// TIA Portal V15.1 export
// export: Created 2024-05-17T05:38:54.7838855Z, ExportSetting WithDefaults, DisplayName Totally Integrated Automation Portal, DisplayVersion V15.1 Update 5, DisplayName TIA Portal Openness, DisplayVersion V15.1 Update 5, DisplayName SINAMICS Startdrive Advanced, DisplayVersion V15.1, DisplayName G130, G150, S120, S150, SINAMICS MV, S210, DisplayVersion V15.1, DisplayName G110M, G120, G120C, G120D, G120P, DisplayVersion V15.1, DisplayName STEP 7 Professional, DisplayVersion V15.1 Update 5, DisplayName STEP 7 Safety, DisplayVersion V15.1, DisplayName WinCC Professional, DisplayVersion V15.1 Update 5, DisplayName SIMATIC Visualization Architect, DisplayVersion V15.1
FUNCTION "209220ZS01Safety" : Void   // FC375, FBD
TITLE = 209220ZS01 Safety
{ S7_Optimized_Access := 'FALSE' }
AUTHOR : VCG
FAMILY : Local
NAME : 610
VERSION : 0.1
// stored: AutoNumber false, IsIECCheckEnabled false, SetENOAutomatically False, UDAEnableTagReadback false
   VAR_OUTPUT
      O_AlarmA : Bool;   // Alarm A
      O_AlarmB : Bool;   // Alarm B
      O_AlarmC : Bool;   // Alarm C
      O_AlarmD : Bool;   // Alarm D
      O_AlarmABCondition : Bool;   // Alarms resetable
      H_IAnim : Word;   // Icon Animation
   END_VAR
BEGIN

REGION Network 1: **** 2.1 - Enable Alarms **** 220CS22M4SG10F & SG11F Check if both safety sensors are activated
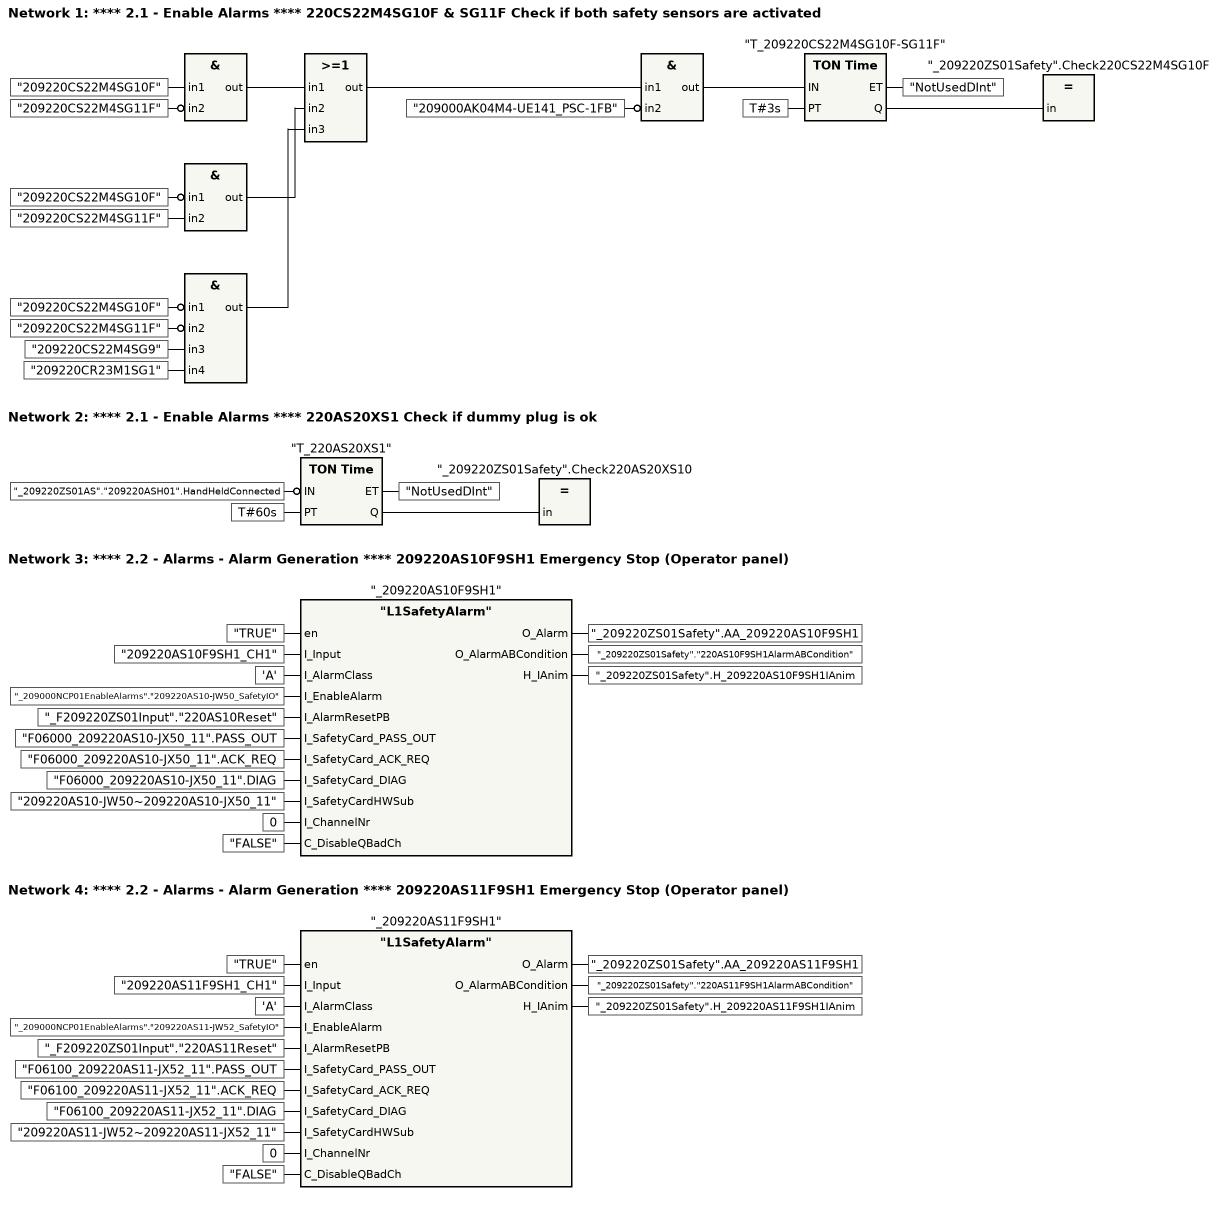
   "T_209220CS22M4SG10F-SG11F".TON(IN := (("209220CS22M4SG10F" AND NOT "209220CS22M4SG11F") OR (NOT "209220CS22M4SG10F" AND "209220CS22M4SG11F") OR (NOT "209220CS22M4SG10F" AND NOT "209220CS22M4SG11F" AND "209220CS22M4SG9" AND "209220CR23M1SG1")) AND NOT "209000AK04M4-UE141_PSC-1FB",
                           PT := T#3s,
                           ET => "NotUsedDInt");
   "_209220ZS01Safety".Check220CS22M4SG10F := "T_209220CS22M4SG10F-SG11F".Q;
END_REGION

REGION Network 2: **** 2.1 - Enable Alarms **** 220AS20XS1 Check if dummy plug is ok
   "T_220AS20XS1".TON(IN := NOT "_209220ZS01AS"."209220ASH01".HandHeldConnected,
                      PT := T#60s,
                      ET => "NotUsedDInt");
   "_209220ZS01Safety".Check220AS20XS10 := "T_220AS20XS1".Q;
END_REGION

REGION Network 3: **** 2.2 - Alarms - Alarm Generation **** 209220AS10F9SH1 Emergency Stop (Operator panel)
   // Emergency Stop
   IF "TRUE" THEN
       "_209220AS10F9SH1"(I_Input := "209220AS10F9SH1_CH1",   // "L1SafetyAlarm"
                          I_AlarmClass := 'A',
                          I_EnableAlarm := "_209000NCP01EnableAlarms"."209220AS10-JW50_SafetyIO",
                          I_AlarmResetPB := "_F209220ZS01Input"."220AS10Reset",
                          I_SafetyCard_PASS_OUT := "F06000_209220AS10-JX50_11".PASS_OUT,
                          I_SafetyCard_ACK_REQ := "F06000_209220AS10-JX50_11".ACK_REQ,
                          I_SafetyCard_DIAG := "F06000_209220AS10-JX50_11".DIAG,
                          I_SafetyCardHWSub := "209220AS10-JW50~209220AS10-JX50_11",
                          I_ChannelNr := 0,
                          C_DisableQBadCh := "FALSE",
                          O_Alarm => "_209220ZS01Safety".AA_209220AS10F9SH1,
                          O_AlarmABCondition => "_209220ZS01Safety"."220AS10F9SH1AlarmABCondition",
                          H_IAnim => "_209220ZS01Safety".H_209220AS10F9SH1IAnim);
   END_IF;
END_REGION

REGION Network 4: **** 2.2 - Alarms - Alarm Generation **** 209220AS11F9SH1 Emergency Stop (Operator panel)
   // Emergency Stop
   IF "TRUE" THEN
       "_209220AS11F9SH1"(I_Input := "209220AS11F9SH1_CH1",   // "L1SafetyAlarm"
                          I_AlarmClass := 'A',
                          I_EnableAlarm := "_209000NCP01EnableAlarms"."209220AS11-JW52_SafetyIO",
                          I_AlarmResetPB := "_F209220ZS01Input"."220AS11Reset",
                          I_SafetyCard_PASS_OUT := "F06100_209220AS11-JX52_11".PASS_OUT,
                          I_SafetyCard_ACK_REQ := "F06100_209220AS11-JX52_11".ACK_REQ,
                          I_SafetyCard_DIAG := "F06100_209220AS11-JX52_11".DIAG,
                          I_SafetyCardHWSub := "209220AS11-JW52~209220AS11-JX52_11",
                          I_ChannelNr := 0,
                          C_DisableQBadCh := "FALSE",
                          O_Alarm => "_209220ZS01Safety".AA_209220AS11F9SH1,
                          O_AlarmABCondition => "_209220ZS01Safety"."220AS11F9SH1AlarmABCondition",
                          H_IAnim => "_209220ZS01Safety".H_209220AS11F9SH1IAnim);
   END_IF;
END_REGION

REGION Network 5: **** 2.2 - Alarms - Alarm Generation **** 209220AS20F9SH1 Emergency Stop (Start/Stop panel)
   // Emergency Stop
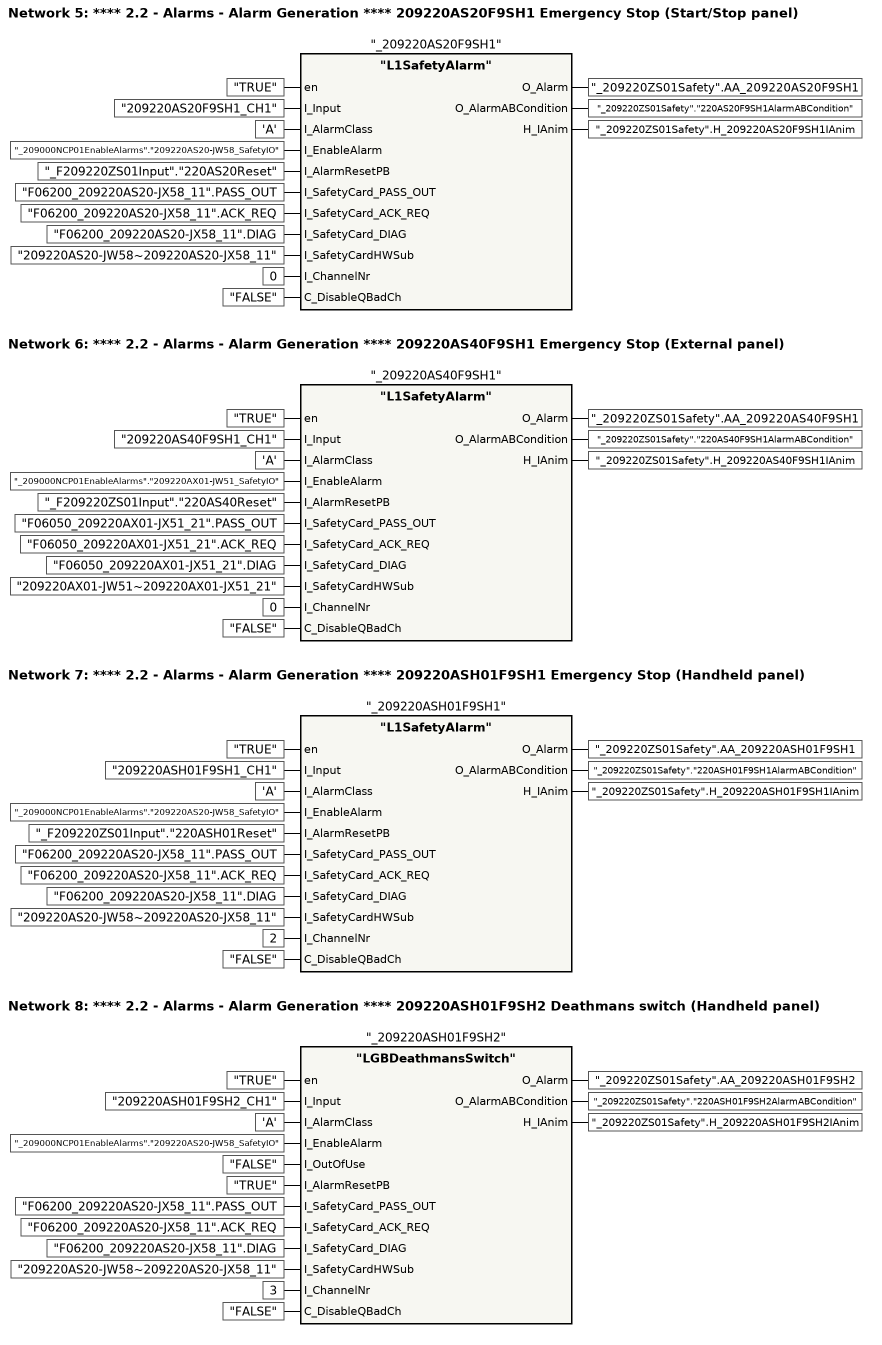
   IF "TRUE" THEN
       "_209220AS20F9SH1"(I_Input := "209220AS20F9SH1_CH1",   // "L1SafetyAlarm"
                          I_AlarmClass := 'A',
                          I_EnableAlarm := "_209000NCP01EnableAlarms"."209220AS20-JW58_SafetyIO",
                          I_AlarmResetPB := "_F209220ZS01Input"."220AS20Reset",
                          I_SafetyCard_PASS_OUT := "F06200_209220AS20-JX58_11".PASS_OUT,
                          I_SafetyCard_ACK_REQ := "F06200_209220AS20-JX58_11".ACK_REQ,
                          I_SafetyCard_DIAG := "F06200_209220AS20-JX58_11".DIAG,
                          I_SafetyCardHWSub := "209220AS20-JW58~209220AS20-JX58_11",
                          I_ChannelNr := 0,
                          C_DisableQBadCh := "FALSE",
                          O_Alarm => "_209220ZS01Safety".AA_209220AS20F9SH1,
                          O_AlarmABCondition => "_209220ZS01Safety"."220AS20F9SH1AlarmABCondition",
                          H_IAnim => "_209220ZS01Safety".H_209220AS20F9SH1IAnim);
   END_IF;
END_REGION

REGION Network 6: **** 2.2 - Alarms - Alarm Generation **** 209220AS40F9SH1 Emergency Stop (External panel)
   // Emergency Stop
   IF "TRUE" THEN
       "_209220AS40F9SH1"(I_Input := "209220AS40F9SH1_CH1",   // "L1SafetyAlarm"
                          I_AlarmClass := 'A',
                          I_EnableAlarm := "_209000NCP01EnableAlarms"."209220AX01-JW51_SafetyIO",
                          I_AlarmResetPB := "_F209220ZS01Input"."220AS40Reset",
                          I_SafetyCard_PASS_OUT := "F06050_209220AX01-JX51_21".PASS_OUT,
                          I_SafetyCard_ACK_REQ := "F06050_209220AX01-JX51_21".ACK_REQ,
                          I_SafetyCard_DIAG := "F06050_209220AX01-JX51_21".DIAG,
                          I_SafetyCardHWSub := "209220AX01-JW51~209220AX01-JX51_21",
                          I_ChannelNr := 0,
                          C_DisableQBadCh := "FALSE",
                          O_Alarm => "_209220ZS01Safety".AA_209220AS40F9SH1,
                          O_AlarmABCondition => "_209220ZS01Safety"."220AS40F9SH1AlarmABCondition",
                          H_IAnim => "_209220ZS01Safety".H_209220AS40F9SH1IAnim);
   END_IF;
END_REGION

REGION Network 7: **** 2.2 - Alarms - Alarm Generation **** 209220ASH01F9SH1 Emergency Stop (Handheld panel)
   // Emergency Stop
   IF "TRUE" THEN
       "_209220ASH01F9SH1"(I_Input := "209220ASH01F9SH1_CH1",   // "L1SafetyAlarm"
                           I_AlarmClass := 'A',
                           I_EnableAlarm := "_209000NCP01EnableAlarms"."209220AS20-JW58_SafetyIO",
                           I_AlarmResetPB := "_F209220ZS01Input"."220ASH01Reset",
                           I_SafetyCard_PASS_OUT := "F06200_209220AS20-JX58_11".PASS_OUT,
                           I_SafetyCard_ACK_REQ := "F06200_209220AS20-JX58_11".ACK_REQ,
                           I_SafetyCard_DIAG := "F06200_209220AS20-JX58_11".DIAG,
                           I_SafetyCardHWSub := "209220AS20-JW58~209220AS20-JX58_11",
                           I_ChannelNr := 2,
                           C_DisableQBadCh := "FALSE",
                           O_Alarm => "_209220ZS01Safety".AA_209220ASH01F9SH1,
                           O_AlarmABCondition => "_209220ZS01Safety"."220ASH01F9SH1AlarmABCondition",
                           H_IAnim => "_209220ZS01Safety".H_209220ASH01F9SH1IAnim);
   END_IF;
END_REGION

REGION Network 8: **** 2.2 - Alarms - Alarm Generation **** 209220ASH01F9SH2 Deathmans switch (Handheld panel)
   // Deathmans switch
   IF "TRUE" THEN
       "_209220ASH01F9SH2"(I_Input := "209220ASH01F9SH2_CH1",   // "LGBDeathmansSwitch"
                           I_AlarmClass := 'A',
                           I_EnableAlarm := "_209000NCP01EnableAlarms"."209220AS20-JW58_SafetyIO",
                           I_OutOfUse := "FALSE",
                           I_AlarmResetPB := "TRUE",
                           I_SafetyCard_PASS_OUT := "F06200_209220AS20-JX58_11".PASS_OUT,
                           I_SafetyCard_ACK_REQ := "F06200_209220AS20-JX58_11".ACK_REQ,
                           I_SafetyCard_DIAG := "F06200_209220AS20-JX58_11".DIAG,
                           I_SafetyCardHWSub := "209220AS20-JW58~209220AS20-JX58_11",
                           I_ChannelNr := 3,
                           C_DisableQBadCh := "FALSE",
                           O_Alarm => "_209220ZS01Safety".AA_209220ASH01F9SH2,
                           O_AlarmABCondition => "_209220ZS01Safety"."220ASH01F9SH2AlarmABCondition",
                           H_IAnim => "_209220ZS01Safety".H_209220ASH01F9SH2IAnim);
   END_IF;
END_REGION

REGION Network 9: **** 2.2 - Alarms - Alarm Generation **** 020R02F9SH / **** 2.2 - Alarms - Alarm Generation **** 209000AK04F9QC1FB Feedback Alarm
   // E-Stop Push Button / Feedback Alarm
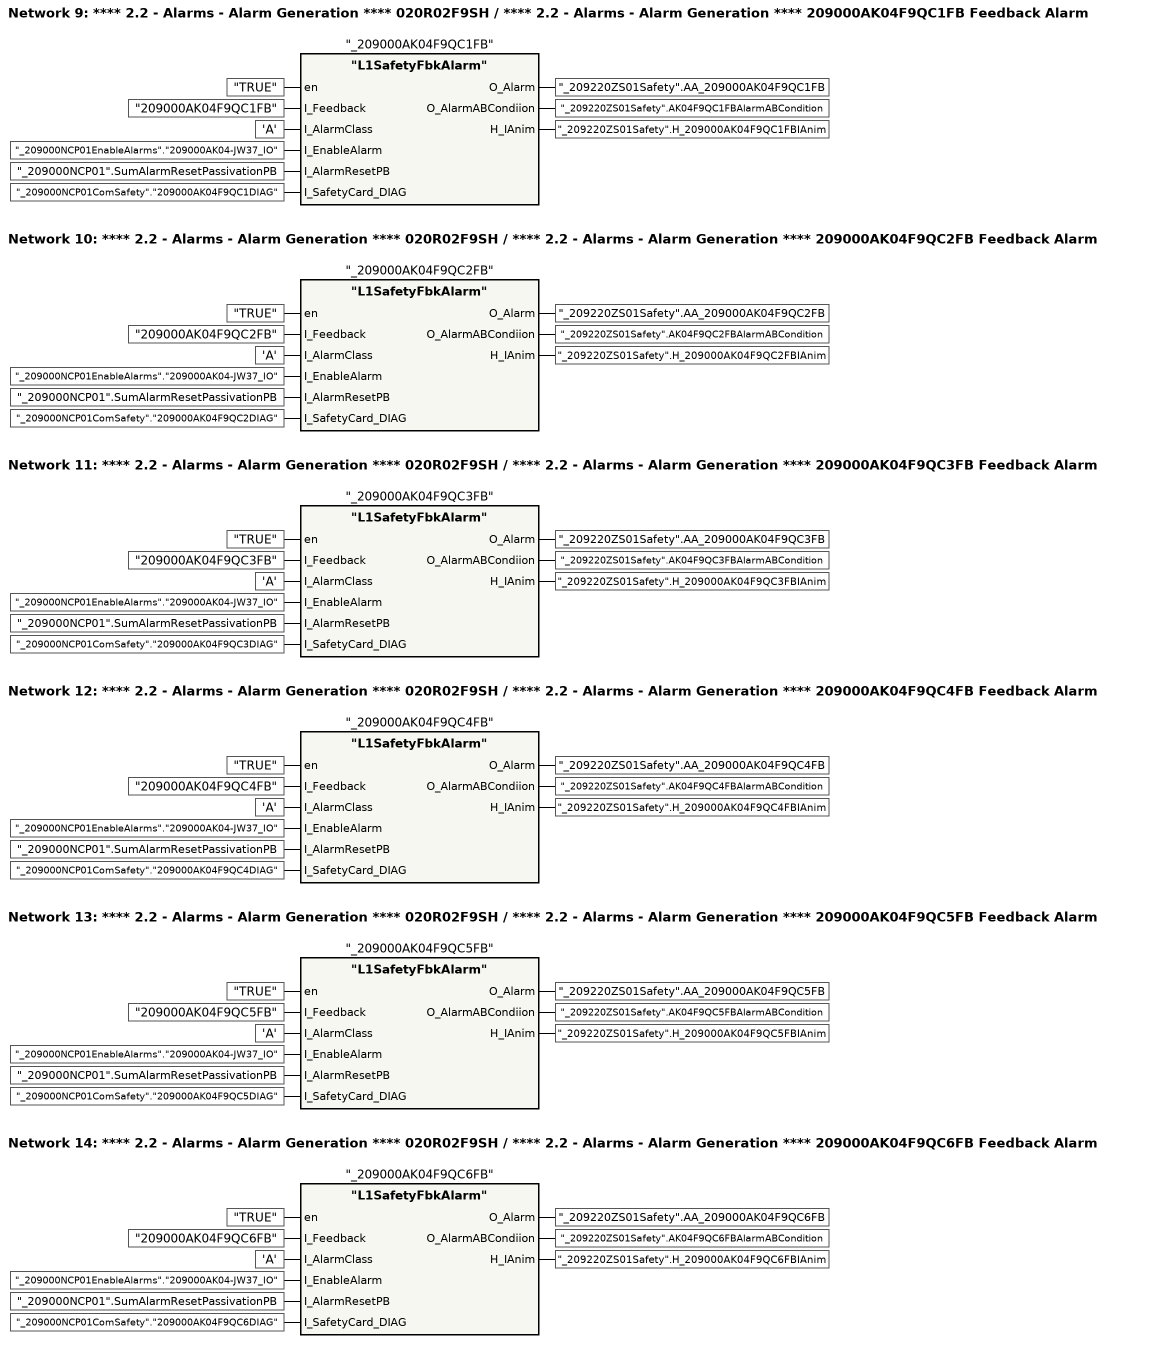
   IF "TRUE" THEN
       "_209000AK04F9QC1FB"(I_Feedback := "209000AK04F9QC1FB",   // "L1SafetyFbkAlarm"
                            I_AlarmClass := 'A',
                            I_EnableAlarm := "_209000NCP01EnableAlarms"."209000AK04-JW37_IO",
                            I_AlarmResetPB := "_209000NCP01".SumAlarmResetPassivationPB,
                            I_SafetyCard_DIAG := "_209000NCP01ComSafety"."209000AK04F9QC1DIAG",
                            O_Alarm => "_209220ZS01Safety".AA_209000AK04F9QC1FB,
                            O_AlarmABCondiion => "_209220ZS01Safety".AK04F9QC1FBAlarmABCondition,
                            H_IAnim => "_209220ZS01Safety".H_209000AK04F9QC1FBIAnim);
   END_IF;
END_REGION

REGION Network 10: **** 2.2 - Alarms - Alarm Generation **** 020R02F9SH / **** 2.2 - Alarms - Alarm Generation **** 209000AK04F9QC2FB Feedback Alarm
   // E-Stop Push Button / Feedback Alarm
   IF "TRUE" THEN
       "_209000AK04F9QC2FB"(I_Feedback := "209000AK04F9QC2FB",   // "L1SafetyFbkAlarm"
                            I_AlarmClass := 'A',
                            I_EnableAlarm := "_209000NCP01EnableAlarms"."209000AK04-JW37_IO",
                            I_AlarmResetPB := "_209000NCP01".SumAlarmResetPassivationPB,
                            I_SafetyCard_DIAG := "_209000NCP01ComSafety"."209000AK04F9QC2DIAG",
                            O_Alarm => "_209220ZS01Safety".AA_209000AK04F9QC2FB,
                            O_AlarmABCondiion => "_209220ZS01Safety".AK04F9QC2FBAlarmABCondition,
                            H_IAnim => "_209220ZS01Safety".H_209000AK04F9QC2FBIAnim);
   END_IF;
END_REGION

REGION Network 11: **** 2.2 - Alarms - Alarm Generation **** 020R02F9SH / **** 2.2 - Alarms - Alarm Generation **** 209000AK04F9QC3FB Feedback Alarm
   // E-Stop Push Button / Feedback Alarm
   IF "TRUE" THEN
       "_209000AK04F9QC3FB"(I_Feedback := "209000AK04F9QC3FB",   // "L1SafetyFbkAlarm"
                            I_AlarmClass := 'A',
                            I_EnableAlarm := "_209000NCP01EnableAlarms"."209000AK04-JW37_IO",
                            I_AlarmResetPB := "_209000NCP01".SumAlarmResetPassivationPB,
                            I_SafetyCard_DIAG := "_209000NCP01ComSafety"."209000AK04F9QC3DIAG",
                            O_Alarm => "_209220ZS01Safety".AA_209000AK04F9QC3FB,
                            O_AlarmABCondiion => "_209220ZS01Safety".AK04F9QC3FBAlarmABCondition,
                            H_IAnim => "_209220ZS01Safety".H_209000AK04F9QC3FBIAnim);
   END_IF;
END_REGION

REGION Network 12: **** 2.2 - Alarms - Alarm Generation **** 020R02F9SH / **** 2.2 - Alarms - Alarm Generation **** 209000AK04F9QC4FB Feedback Alarm
   // E-Stop Push Button / Feedback Alarm
   IF "TRUE" THEN
       "_209000AK04F9QC4FB"(I_Feedback := "209000AK04F9QC4FB",   // "L1SafetyFbkAlarm"
                            I_AlarmClass := 'A',
                            I_EnableAlarm := "_209000NCP01EnableAlarms"."209000AK04-JW37_IO",
                            I_AlarmResetPB := "_209000NCP01".SumAlarmResetPassivationPB,
                            I_SafetyCard_DIAG := "_209000NCP01ComSafety"."209000AK04F9QC4DIAG",
                            O_Alarm => "_209220ZS01Safety".AA_209000AK04F9QC4FB,
                            O_AlarmABCondiion => "_209220ZS01Safety".AK04F9QC4FBAlarmABCondition,
                            H_IAnim => "_209220ZS01Safety".H_209000AK04F9QC4FBIAnim);
   END_IF;
END_REGION

REGION Network 13: **** 2.2 - Alarms - Alarm Generation **** 020R02F9SH / **** 2.2 - Alarms - Alarm Generation **** 209000AK04F9QC5FB Feedback Alarm
   // E-Stop Push Button / Feedback Alarm
   IF "TRUE" THEN
       "_209000AK04F9QC5FB"(I_Feedback := "209000AK04F9QC5FB",   // "L1SafetyFbkAlarm"
                            I_AlarmClass := 'A',
                            I_EnableAlarm := "_209000NCP01EnableAlarms"."209000AK04-JW37_IO",
                            I_AlarmResetPB := "_209000NCP01".SumAlarmResetPassivationPB,
                            I_SafetyCard_DIAG := "_209000NCP01ComSafety"."209000AK04F9QC5DIAG",
                            O_Alarm => "_209220ZS01Safety".AA_209000AK04F9QC5FB,
                            O_AlarmABCondiion => "_209220ZS01Safety".AK04F9QC5FBAlarmABCondition,
                            H_IAnim => "_209220ZS01Safety".H_209000AK04F9QC5FBIAnim);
   END_IF;
END_REGION

REGION Network 14: **** 2.2 - Alarms - Alarm Generation **** 020R02F9SH / **** 2.2 - Alarms - Alarm Generation **** 209000AK04F9QC6FB Feedback Alarm
   // E-Stop Push Button / Feedback Alarm
   IF "TRUE" THEN
       "_209000AK04F9QC6FB"(I_Feedback := "209000AK04F9QC6FB",   // "L1SafetyFbkAlarm"
                            I_AlarmClass := 'A',
                            I_EnableAlarm := "_209000NCP01EnableAlarms"."209000AK04-JW37_IO",
                            I_AlarmResetPB := "_209000NCP01".SumAlarmResetPassivationPB,
                            I_SafetyCard_DIAG := "_209000NCP01ComSafety"."209000AK04F9QC6DIAG",
                            O_Alarm => "_209220ZS01Safety".AA_209000AK04F9QC6FB,
                            O_AlarmABCondiion => "_209220ZS01Safety".AK04F9QC6FBAlarmABCondition,
                            H_IAnim => "_209220ZS01Safety".H_209000AK04F9QC6FBIAnim);
   END_IF;
END_REGION

REGION Network 15: **** 2.2 - Alarms - Alarm Generation **** 209220CHB21M14SG1F Safety sensor
   // Safety sensor
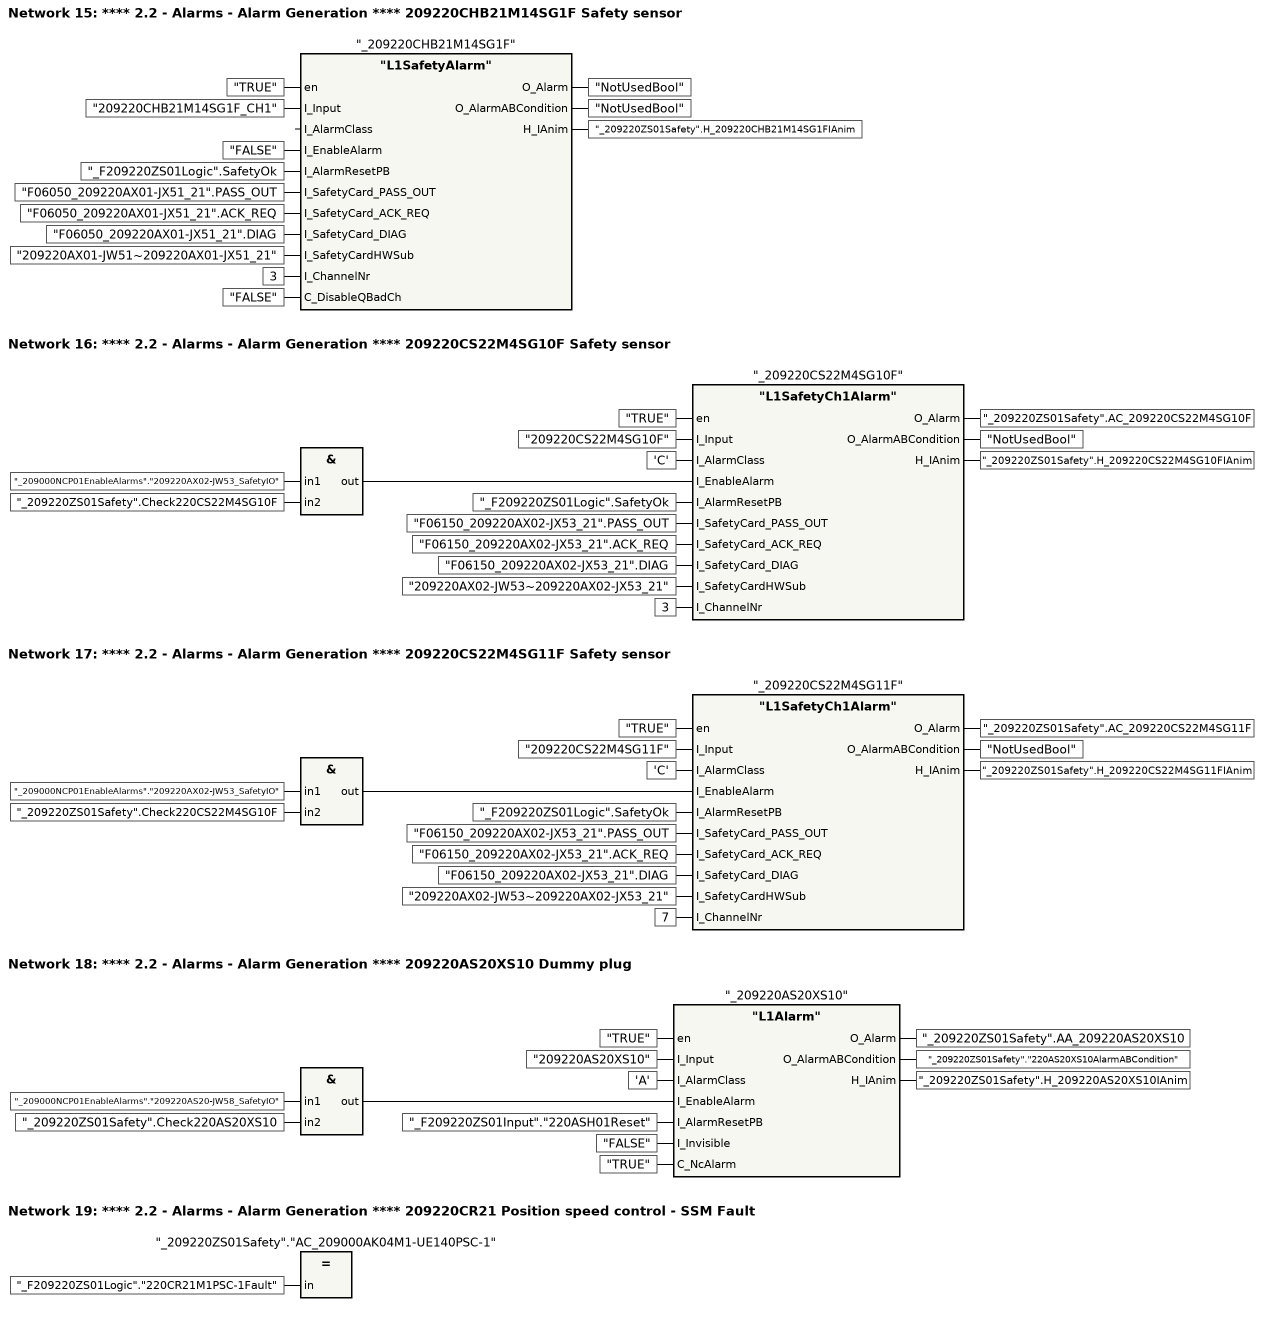
   IF "TRUE" THEN
       "_209220CHB21M14SG1F"(I_Input := "209220CHB21M14SG1F_CH1",   // "L1SafetyAlarm"
                             I_EnableAlarm := "FALSE",
                             I_AlarmResetPB := "_F209220ZS01Logic".SafetyOk,
                             I_SafetyCard_PASS_OUT := "F06050_209220AX01-JX51_21".PASS_OUT,
                             I_SafetyCard_ACK_REQ := "F06050_209220AX01-JX51_21".ACK_REQ,
                             I_SafetyCard_DIAG := "F06050_209220AX01-JX51_21".DIAG,
                             I_SafetyCardHWSub := "209220AX01-JW51~209220AX01-JX51_21",
                             I_ChannelNr := 3,
                             C_DisableQBadCh := "FALSE",
                             O_Alarm => "NotUsedBool",
                             O_AlarmABCondition => "NotUsedBool",
                             H_IAnim => "_209220ZS01Safety".H_209220CHB21M14SG1FIAnim);
   END_IF;
END_REGION

REGION Network 16: **** 2.2 - Alarms - Alarm Generation **** 209220CS22M4SG10F Safety sensor
   // Safety sensor
   IF "TRUE" THEN
       "_209220CS22M4SG10F"(I_Input := "209220CS22M4SG10F",   // "L1SafetyCh1Alarm"
                            I_AlarmClass := 'C',
                            I_EnableAlarm := "_209000NCP01EnableAlarms"."209220AX02-JW53_SafetyIO" AND "_209220ZS01Safety".Check220CS22M4SG10F,
                            I_AlarmResetPB := "_F209220ZS01Logic".SafetyOk,
                            I_SafetyCard_PASS_OUT := "F06150_209220AX02-JX53_21".PASS_OUT,
                            I_SafetyCard_ACK_REQ := "F06150_209220AX02-JX53_21".ACK_REQ,
                            I_SafetyCard_DIAG := "F06150_209220AX02-JX53_21".DIAG,
                            I_SafetyCardHWSub := "209220AX02-JW53~209220AX02-JX53_21",
                            I_ChannelNr := 3,
                            O_Alarm => "_209220ZS01Safety".AC_209220CS22M4SG10F,
                            O_AlarmABCondition => "NotUsedBool",
                            H_IAnim => "_209220ZS01Safety".H_209220CS22M4SG10FIAnim);
   END_IF;
END_REGION

REGION Network 17: **** 2.2 - Alarms - Alarm Generation **** 209220CS22M4SG11F Safety sensor
   // Safety sensor
   IF "TRUE" THEN
       "_209220CS22M4SG11F"(I_Input := "209220CS22M4SG11F",   // "L1SafetyCh1Alarm"
                            I_AlarmClass := 'C',
                            I_EnableAlarm := "_209000NCP01EnableAlarms"."209220AX02-JW53_SafetyIO" AND "_209220ZS01Safety".Check220CS22M4SG10F,
                            I_AlarmResetPB := "_F209220ZS01Logic".SafetyOk,
                            I_SafetyCard_PASS_OUT := "F06150_209220AX02-JX53_21".PASS_OUT,
                            I_SafetyCard_ACK_REQ := "F06150_209220AX02-JX53_21".ACK_REQ,
                            I_SafetyCard_DIAG := "F06150_209220AX02-JX53_21".DIAG,
                            I_SafetyCardHWSub := "209220AX02-JW53~209220AX02-JX53_21",
                            I_ChannelNr := 7,
                            O_Alarm => "_209220ZS01Safety".AC_209220CS22M4SG11F,
                            O_AlarmABCondition => "NotUsedBool",
                            H_IAnim => "_209220ZS01Safety".H_209220CS22M4SG11FIAnim);
   END_IF;
END_REGION

REGION Network 18: **** 2.2 - Alarms - Alarm Generation **** 209220AS20XS10 Dummy plug
   IF "TRUE" THEN
       "_209220AS20XS10"(I_Input := "209220AS20XS10",   // "L1Alarm"
                         I_AlarmClass := 'A',
                         I_EnableAlarm := "_209000NCP01EnableAlarms"."209220AS20-JW58_SafetyIO" AND "_209220ZS01Safety".Check220AS20XS10,
                         I_AlarmResetPB := "_F209220ZS01Input"."220ASH01Reset",
                         I_Invisible := "FALSE",
                         C_NcAlarm := "TRUE",
                         O_Alarm => "_209220ZS01Safety".AA_209220AS20XS10,
                         O_AlarmABCondition => "_209220ZS01Safety"."220AS20XS10AlarmABCondition",
                         H_IAnim => "_209220ZS01Safety".H_209220AS20XS10IAnim);
   END_IF;
END_REGION

REGION Network 19: **** 2.2 - Alarms - Alarm Generation **** 209220CR21 Position speed control - SSM Fault
   // SEW Safety Function
   "_209220ZS01Safety"."AC_209000AK04M1-UE140PSC-1" := "_F209220ZS01Logic"."220CR21M1PSC-1Fault";
END_REGION

REGION Network 20: **** 2.2 - Alarms - Alarm Generation **** 209220CS22 Position speed control - SSM Fault
   // SEW Safety Function
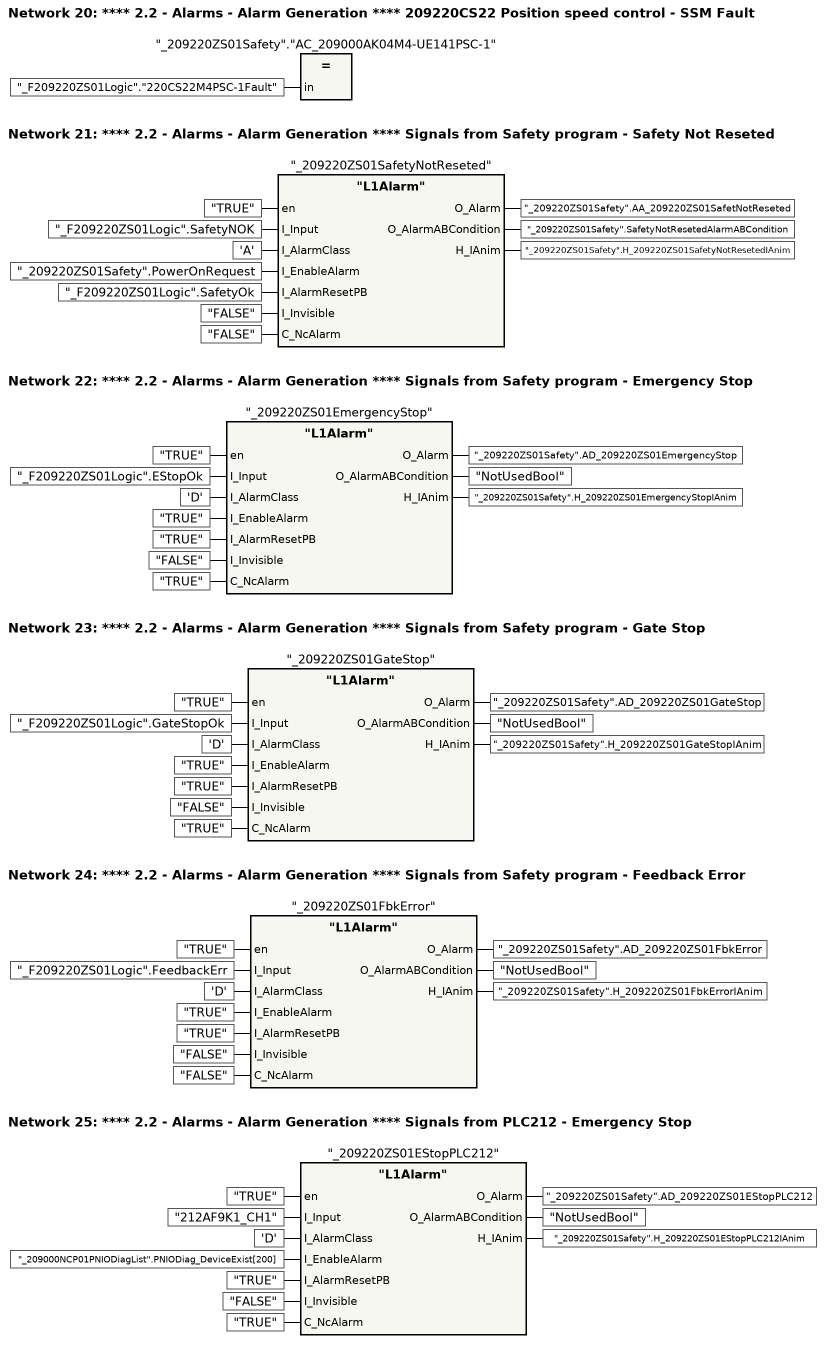
   "_209220ZS01Safety"."AC_209000AK04M4-UE141PSC-1" := "_F209220ZS01Logic"."220CS22M4PSC-1Fault";
END_REGION

REGION Network 21: **** 2.2 - Alarms - Alarm Generation **** Signals from Safety program - Safety Not Reseted
   // Safety Has Not Been Reseted
   IF "TRUE" THEN
       "_209220ZS01SafetyNotReseted"(I_Input := "_F209220ZS01Logic".SafetyNOK,   // "L1Alarm"
                               I_AlarmClass := 'A',
                               I_EnableAlarm := "_209220ZS01Safety".PowerOnRequest,
                               I_AlarmResetPB := "_F209220ZS01Logic".SafetyOk,
                               I_Invisible := "FALSE",
                               C_NcAlarm := "FALSE",
                               O_Alarm => "_209220ZS01Safety".AA_209220ZS01SafetNotReseted,
                               O_AlarmABCondition => "_209220ZS01Safety".SafetyNotResetedAlarmABCondition,
                               H_IAnim => "_209220ZS01Safety".H_209220ZS01SafetyNotResetedIAnim);
   END_IF;
END_REGION

REGION Network 22: **** 2.2 - Alarms - Alarm Generation **** Signals from Safety program - Emergency Stop
   // Emergency Stop
   IF "TRUE" THEN
       "_209220ZS01EmergencyStop"(I_Input := "_F209220ZS01Logic".EStopOk,   // "L1Alarm"
                               I_AlarmClass := 'D',
                               I_EnableAlarm := "TRUE",
                               I_AlarmResetPB := "TRUE",
                               I_Invisible := "FALSE",
                               C_NcAlarm := "TRUE",
                               O_Alarm => "_209220ZS01Safety".AD_209220ZS01EmergencyStop,
                               O_AlarmABCondition => "NotUsedBool",
                               H_IAnim => "_209220ZS01Safety".H_209220ZS01EmergencyStopIAnim);
   END_IF;
END_REGION

REGION Network 23: **** 2.2 - Alarms - Alarm Generation **** Signals from Safety program - Gate Stop
   // Gate Stop
   IF "TRUE" THEN
       "_209220ZS01GateStop"(I_Input := "_F209220ZS01Logic".GateStopOk,   // "L1Alarm"
                             I_AlarmClass := 'D',
                             I_EnableAlarm := "TRUE",
                             I_AlarmResetPB := "TRUE",
                             I_Invisible := "FALSE",
                             C_NcAlarm := "TRUE",
                             O_Alarm => "_209220ZS01Safety".AD_209220ZS01GateStop,
                             O_AlarmABCondition => "NotUsedBool",
                             H_IAnim => "_209220ZS01Safety".H_209220ZS01GateStopIAnim);
   END_IF;
END_REGION

REGION Network 24: **** 2.2 - Alarms - Alarm Generation **** Signals from Safety program - Feedback Error
   // Feedback Error
   IF "TRUE" THEN
       "_209220ZS01FbkError"(I_Input := "_F209220ZS01Logic".FeedbackErr,   // "L1Alarm"
                             I_AlarmClass := 'D',
                             I_EnableAlarm := "TRUE",
                             I_AlarmResetPB := "TRUE",
                             I_Invisible := "FALSE",
                             C_NcAlarm := "FALSE",
                             O_Alarm => "_209220ZS01Safety".AD_209220ZS01FbkError,
                             O_AlarmABCondition => "NotUsedBool",
                             H_IAnim => "_209220ZS01Safety".H_209220ZS01FbkErrorIAnim);
   END_IF;
END_REGION

REGION Network 25: **** 2.2 - Alarms - Alarm Generation **** Signals from PLC212 - Emergency Stop
   IF "TRUE" THEN
       "_209220ZS01EStopPLC212"(I_Input := "212AF9K1_CH1",   // "L1Alarm"
                               I_AlarmClass := 'D',
                               I_EnableAlarm := "_209000NCP01PNIODiagList".PNIODiag_DeviceExist[200],
                               I_AlarmResetPB := "TRUE",
                               I_Invisible := "FALSE",
                               C_NcAlarm := "TRUE",
                               O_Alarm => "_209220ZS01Safety".AD_209220ZS01EStopPLC212,
                               O_AlarmABCondition => "NotUsedBool",
                               H_IAnim => "_209220ZS01Safety".H_209220ZS01EStopPLC212IAnim);
   END_IF;
END_REGION

REGION Network 26: **** 2.2 - Alarms - Alarm Generation **** Signals from PLC212 - Motion Stop 220CR23 & 220CS22
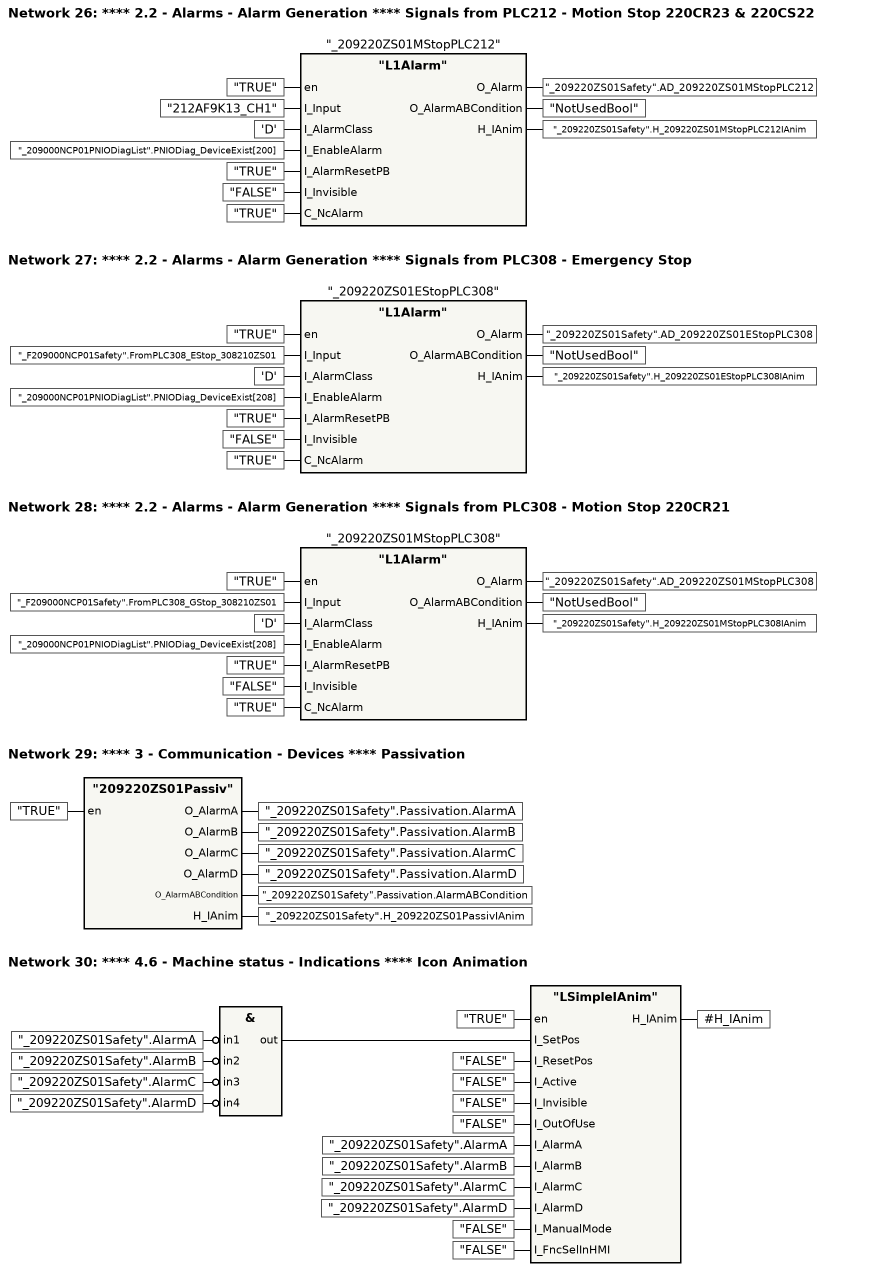
   IF "TRUE" THEN
       "_209220ZS01MStopPLC212"(I_Input := "212AF9K13_CH1",   // "L1Alarm"
                               I_AlarmClass := 'D',
                               I_EnableAlarm := "_209000NCP01PNIODiagList".PNIODiag_DeviceExist[200],
                               I_AlarmResetPB := "TRUE",
                               I_Invisible := "FALSE",
                               C_NcAlarm := "TRUE",
                               O_Alarm => "_209220ZS01Safety".AD_209220ZS01MStopPLC212,
                               O_AlarmABCondition => "NotUsedBool",
                               H_IAnim => "_209220ZS01Safety".H_209220ZS01MStopPLC212IAnim);
   END_IF;
END_REGION

REGION Network 27: **** 2.2 - Alarms - Alarm Generation **** Signals from PLC308 - Emergency Stop
   IF "TRUE" THEN
       "_209220ZS01EStopPLC308"(I_Input := "_F209000NCP01Safety".FromPLC308_EStop_308210ZS01,   // "L1Alarm"
                               I_AlarmClass := 'D',
                               I_EnableAlarm := "_209000NCP01PNIODiagList".PNIODiag_DeviceExist[208],
                               I_AlarmResetPB := "TRUE",
                               I_Invisible := "FALSE",
                               C_NcAlarm := "TRUE",
                               O_Alarm => "_209220ZS01Safety".AD_209220ZS01EStopPLC308,
                               O_AlarmABCondition => "NotUsedBool",
                               H_IAnim => "_209220ZS01Safety".H_209220ZS01EStopPLC308IAnim);
   END_IF;
END_REGION

REGION Network 28: **** 2.2 - Alarms - Alarm Generation **** Signals from PLC308 - Motion Stop 220CR21
   IF "TRUE" THEN
       "_209220ZS01MStopPLC308"(I_Input := "_F209000NCP01Safety".FromPLC308_GStop_308210ZS01,   // "L1Alarm"
                               I_AlarmClass := 'D',
                               I_EnableAlarm := "_209000NCP01PNIODiagList".PNIODiag_DeviceExist[208],
                               I_AlarmResetPB := "TRUE",
                               I_Invisible := "FALSE",
                               C_NcAlarm := "TRUE",
                               O_Alarm => "_209220ZS01Safety".AD_209220ZS01MStopPLC308,
                               O_AlarmABCondition => "NotUsedBool",
                               H_IAnim => "_209220ZS01Safety".H_209220ZS01MStopPLC308IAnim);
   END_IF;
END_REGION

REGION Network 29: **** 3 - Communication - Devices **** Passivation
   // Passivation
   IF "TRUE" THEN
       "209220ZS01Passiv"(O_AlarmA => "_209220ZS01Safety".Passivation.AlarmA,
                          O_AlarmB => "_209220ZS01Safety".Passivation.AlarmB,
                          O_AlarmC => "_209220ZS01Safety".Passivation.AlarmC,
                          O_AlarmD => "_209220ZS01Safety".Passivation.AlarmD,
                          O_AlarmABCondition => "_209220ZS01Safety".Passivation.AlarmABCondition,
                          H_IAnim => "_209220ZS01Safety".H_209220ZS01PassivIAnim);
   END_IF;
END_REGION

REGION Network 30: **** 4.6 - Machine status - Indications **** Icon Animation
   // Icon animation
   IF "TRUE" THEN
       "LSimpleIAnim"(I_SetPos := NOT "_209220ZS01Safety".AlarmA AND NOT "_209220ZS01Safety".AlarmB AND NOT "_209220ZS01Safety".AlarmC AND NOT "_209220ZS01Safety".AlarmD,
                      I_ResetPos := "FALSE",
                      I_Active := "FALSE",
                      I_Invisible := "FALSE",
                      I_OutOfUse := "FALSE",
                      I_AlarmA := "_209220ZS01Safety".AlarmA,
                      I_AlarmB := "_209220ZS01Safety".AlarmB,
                      I_AlarmC := "_209220ZS01Safety".AlarmC,
                      I_AlarmD := "_209220ZS01Safety".AlarmD,
                      I_ManualMode := "FALSE",
                      I_FncSelInHMI := "FALSE",
                      H_IAnim => #H_IAnim);
   END_IF;
END_REGION

REGION Network 31: **** 4.6 - Machine status - Indications **** Animation
   // Animation
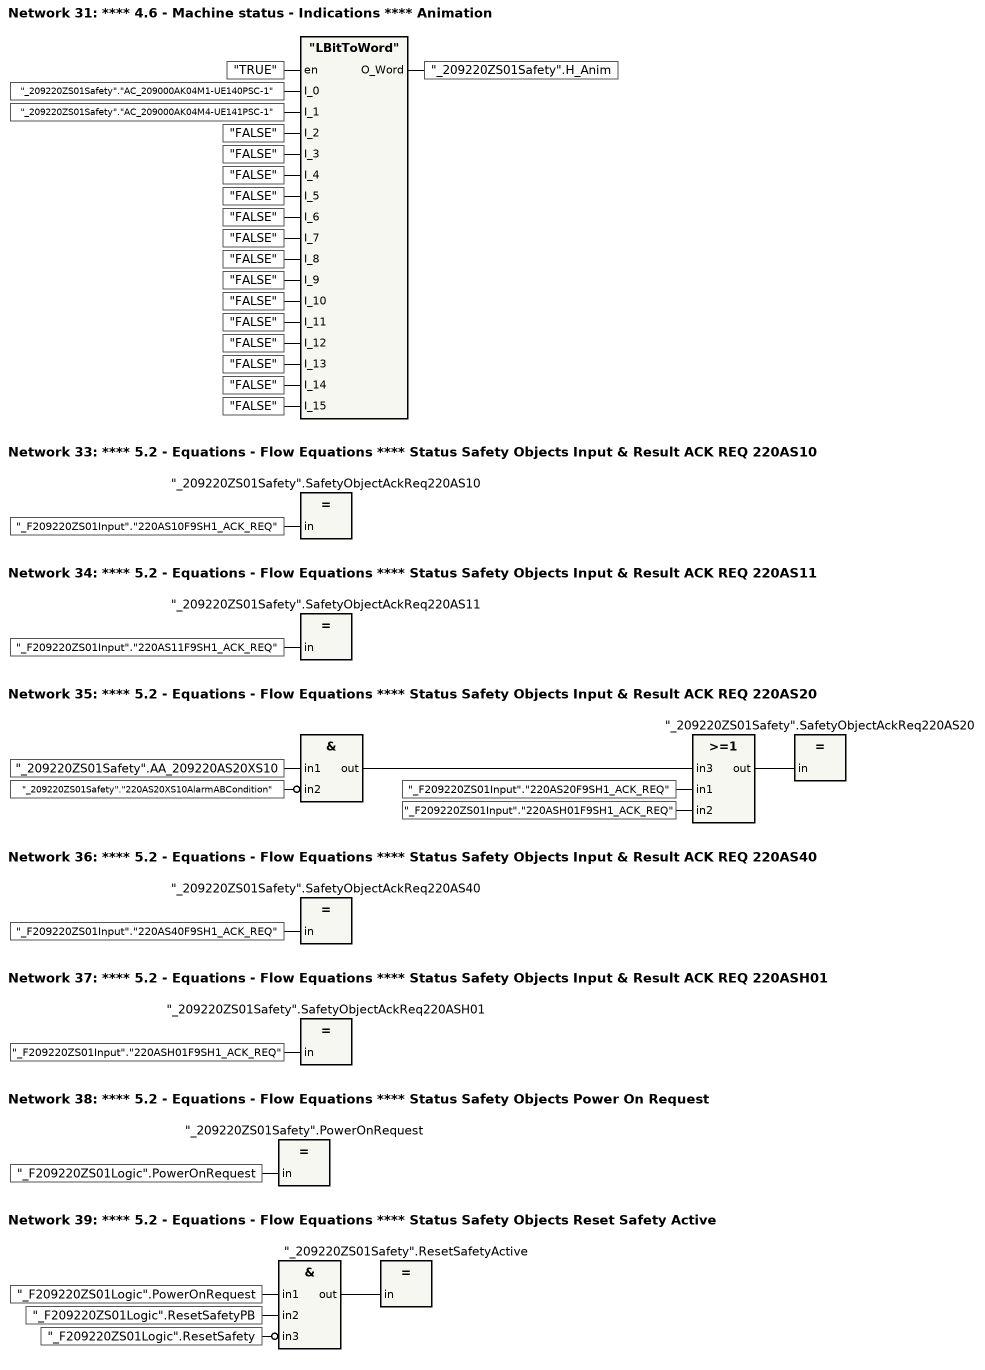
   IF "TRUE" THEN
       "LBitToWord"(I_0 := "_209220ZS01Safety"."AC_209000AK04M1-UE140PSC-1",
                    I_1 := "_209220ZS01Safety"."AC_209000AK04M4-UE141PSC-1",
                    I_2 := "FALSE",
                    I_3 := "FALSE",
                    I_4 := "FALSE",
                    I_5 := "FALSE",
                    I_6 := "FALSE",
                    I_7 := "FALSE",
                    I_8 := "FALSE",
                    I_9 := "FALSE",
                    I_10 := "FALSE",
                    I_11 := "FALSE",
                    I_12 := "FALSE",
                    I_13 := "FALSE",
                    I_14 := "FALSE",
                    I_15 := "FALSE",
                    O_Word => "_209220ZS01Safety".H_Anim);
   END_IF;
END_REGION

NETWORK
TITLE = **** 4.6 - Machine Status - Indications **** Animation DB number
// DB number
      OPN   "_209220ZS01Safety";
      L     DBNO;
      T     "_209220ZS01Safety".H_DBnr;

REGION Network 33: **** 5.2 - Equations - Flow Equations **** Status Safety Objects Input & Result ACK REQ 220AS10
   "_209220ZS01Safety".SafetyObjectAckReq220AS10 := "_F209220ZS01Input"."220AS10F9SH1_ACK_REQ";
END_REGION

REGION Network 34: **** 5.2 - Equations - Flow Equations **** Status Safety Objects Input & Result ACK REQ 220AS11
   "_209220ZS01Safety".SafetyObjectAckReq220AS11 := "_F209220ZS01Input"."220AS11F9SH1_ACK_REQ";
END_REGION

REGION Network 35: **** 5.2 - Equations - Flow Equations **** Status Safety Objects Input & Result ACK REQ 220AS20
   "_209220ZS01Safety".SafetyObjectAckReq220AS20 := ("_209220ZS01Safety".AA_209220AS20XS10 AND NOT "_209220ZS01Safety"."220AS20XS10AlarmABCondition") OR "_F209220ZS01Input"."220AS20F9SH1_ACK_REQ" OR "_F209220ZS01Input"."220ASH01F9SH1_ACK_REQ";
END_REGION

REGION Network 36: **** 5.2 - Equations - Flow Equations **** Status Safety Objects Input & Result ACK REQ 220AS40
   "_209220ZS01Safety".SafetyObjectAckReq220AS40 := "_F209220ZS01Input"."220AS40F9SH1_ACK_REQ";
END_REGION

REGION Network 37: **** 5.2 - Equations - Flow Equations **** Status Safety Objects Input & Result ACK REQ 220ASH01
   "_209220ZS01Safety".SafetyObjectAckReq220ASH01 := "_F209220ZS01Input"."220ASH01F9SH1_ACK_REQ";
END_REGION

REGION Network 38: **** 5.2 - Equations - Flow Equations **** Status Safety Objects Power On Request
   "_209220ZS01Safety".PowerOnRequest := "_F209220ZS01Logic".PowerOnRequest;
END_REGION

REGION Network 39: **** 5.2 - Equations - Flow Equations **** Status Safety Objects Reset Safety Active
   "_209220ZS01Safety".ResetSafetyActive := "_F209220ZS01Logic".PowerOnRequest AND "_F209220ZS01Logic".ResetSafetyPB AND NOT "_F209220ZS01Logic".ResetSafety;
END_REGION

REGION Network 40: **** 5.2 - Equations - Flow Equations **** Feedback Error
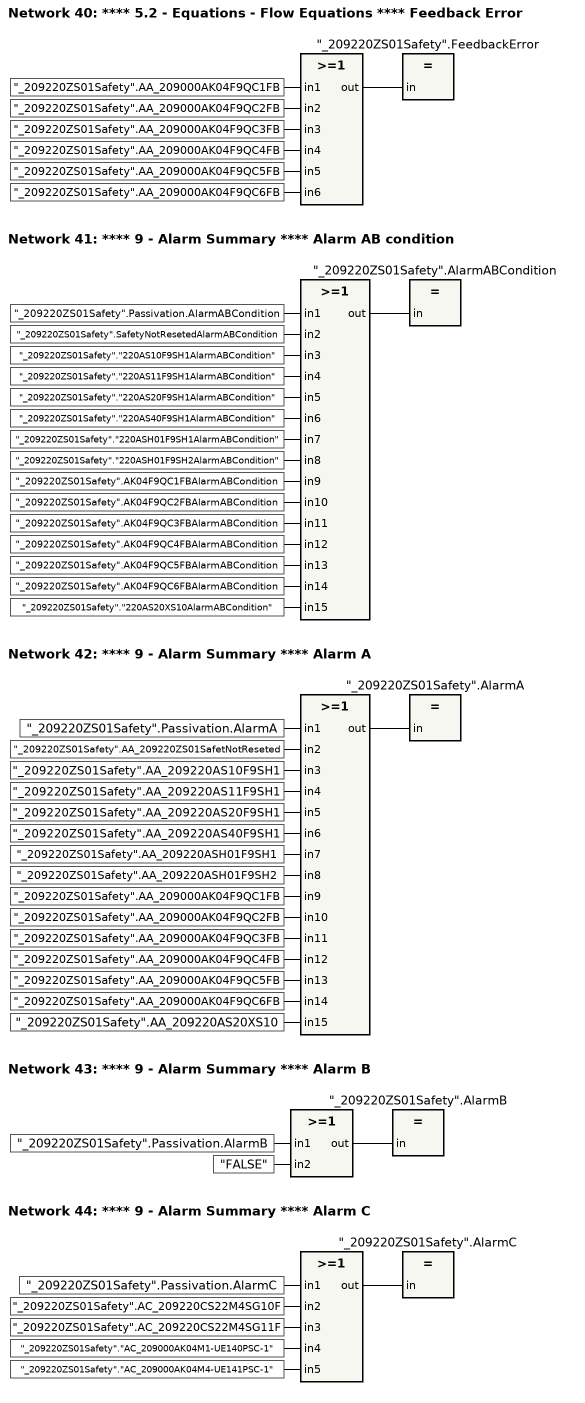
   "_209220ZS01Safety".FeedbackError := "_209220ZS01Safety".AA_209000AK04F9QC1FB OR "_209220ZS01Safety".AA_209000AK04F9QC2FB OR "_209220ZS01Safety".AA_209000AK04F9QC3FB OR "_209220ZS01Safety".AA_209000AK04F9QC4FB OR "_209220ZS01Safety".AA_209000AK04F9QC5FB OR "_209220ZS01Safety".AA_209000AK04F9QC6FB;
END_REGION

REGION Network 41: **** 9 - Alarm Summary **** Alarm AB condition
   // Alarm AB condition
   "_209220ZS01Safety".AlarmABCondition := "_209220ZS01Safety".Passivation.AlarmABCondition OR "_209220ZS01Safety".SafetyNotResetedAlarmABCondition OR "_209220ZS01Safety"."220AS10F9SH1AlarmABCondition" OR "_209220ZS01Safety"."220AS11F9SH1AlarmABCondition" OR "_209220ZS01Safety"."220AS20F9SH1AlarmABCondition" OR "_209220ZS01Safety"."220AS40F9SH1AlarmABCondition" OR "_209220ZS01Safety"."220ASH01F9SH1AlarmABCondition" OR "_209220ZS01Safety"."220ASH01F9SH2AlarmABCondition" OR "_209220ZS01Safety".AK04F9QC1FBAlarmABCondition OR "_209220ZS01Safety".AK04F9QC2FBAlarmABCondition OR "_209220ZS01Safety".AK04F9QC3FBAlarmABCondition OR "_209220ZS01Safety".AK04F9QC4FBAlarmABCondition OR "_209220ZS01Safety".AK04F9QC5FBAlarmABCondition OR "_209220ZS01Safety".AK04F9QC6FBAlarmABCondition OR "_209220ZS01Safety"."220AS20XS10AlarmABCondition";
END_REGION

REGION Network 42: **** 9 - Alarm Summary **** Alarm A
   // Summary of alarms A
   "_209220ZS01Safety".AlarmA := "_209220ZS01Safety".Passivation.AlarmA OR "_209220ZS01Safety".AA_209220ZS01SafetNotReseted OR "_209220ZS01Safety".AA_209220AS10F9SH1 OR "_209220ZS01Safety".AA_209220AS11F9SH1 OR "_209220ZS01Safety".AA_209220AS20F9SH1 OR "_209220ZS01Safety".AA_209220AS40F9SH1 OR "_209220ZS01Safety".AA_209220ASH01F9SH1 OR "_209220ZS01Safety".AA_209220ASH01F9SH2 OR "_209220ZS01Safety".AA_209000AK04F9QC1FB OR "_209220ZS01Safety".AA_209000AK04F9QC2FB OR "_209220ZS01Safety".AA_209000AK04F9QC3FB OR "_209220ZS01Safety".AA_209000AK04F9QC4FB OR "_209220ZS01Safety".AA_209000AK04F9QC5FB OR "_209220ZS01Safety".AA_209000AK04F9QC6FB OR "_209220ZS01Safety".AA_209220AS20XS10;
END_REGION

REGION Network 43: **** 9 - Alarm Summary **** Alarm B
   // Summary of alarms B
   "_209220ZS01Safety".AlarmB := "_209220ZS01Safety".Passivation.AlarmB OR "FALSE";
END_REGION

REGION Network 44: **** 9 - Alarm Summary **** Alarm C
   // Summary of alarms C
   "_209220ZS01Safety".AlarmC := "_209220ZS01Safety".Passivation.AlarmC OR "_209220ZS01Safety".AC_209220CS22M4SG10F OR "_209220ZS01Safety".AC_209220CS22M4SG11F OR "_209220ZS01Safety"."AC_209000AK04M1-UE140PSC-1" OR "_209220ZS01Safety"."AC_209000AK04M4-UE141PSC-1";
END_REGION

REGION Network 45: **** 9 - Alarm Summary **** Alarm D
   // Summary of alarms D
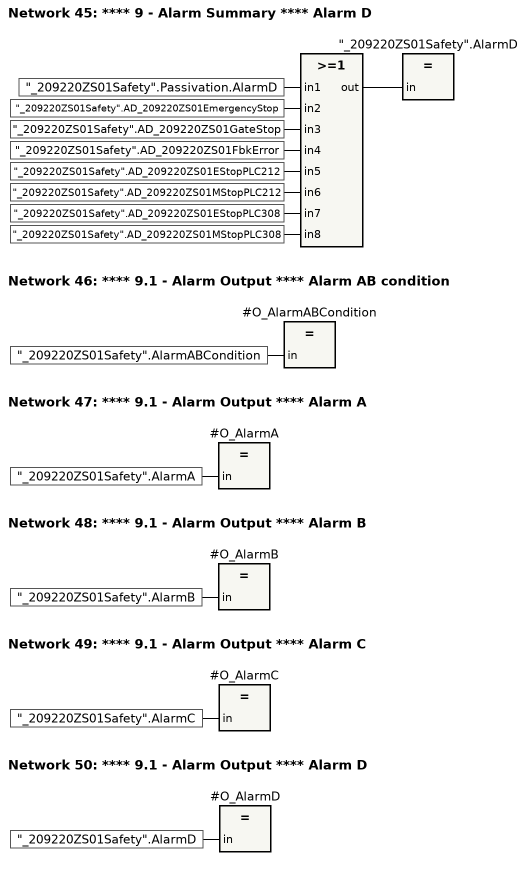
   "_209220ZS01Safety".AlarmD := "_209220ZS01Safety".Passivation.AlarmD OR "_209220ZS01Safety".AD_209220ZS01EmergencyStop OR "_209220ZS01Safety".AD_209220ZS01GateStop OR "_209220ZS01Safety".AD_209220ZS01FbkError OR "_209220ZS01Safety".AD_209220ZS01EStopPLC212 OR "_209220ZS01Safety".AD_209220ZS01MStopPLC212 OR "_209220ZS01Safety".AD_209220ZS01EStopPLC308 OR "_209220ZS01Safety".AD_209220ZS01MStopPLC308;
END_REGION

REGION Network 46: **** 9.1 - Alarm Output **** Alarm AB condition
   // Alarm AB condition
   #O_AlarmABCondition := "_209220ZS01Safety".AlarmABCondition;
END_REGION

REGION Network 47: **** 9.1 - Alarm Output **** Alarm A
   // Summary of alarms A
   #O_AlarmA := "_209220ZS01Safety".AlarmA;
END_REGION

REGION Network 48: **** 9.1 - Alarm Output **** Alarm B
   // Summary of alarms B
   #O_AlarmB := "_209220ZS01Safety".AlarmB;
END_REGION

REGION Network 49: **** 9.1 - Alarm Output **** Alarm C
   // Summary of alarms C
   #O_AlarmC := "_209220ZS01Safety".AlarmC;
END_REGION

REGION Network 50: **** 9.1 - Alarm Output **** Alarm D
   // Summary of alarms D
   #O_AlarmD := "_209220ZS01Safety".AlarmD;
END_REGION

REGION Network 51: **** 9.2 - Alarm DWord**** Alarm To DWord
   // Alarm Word
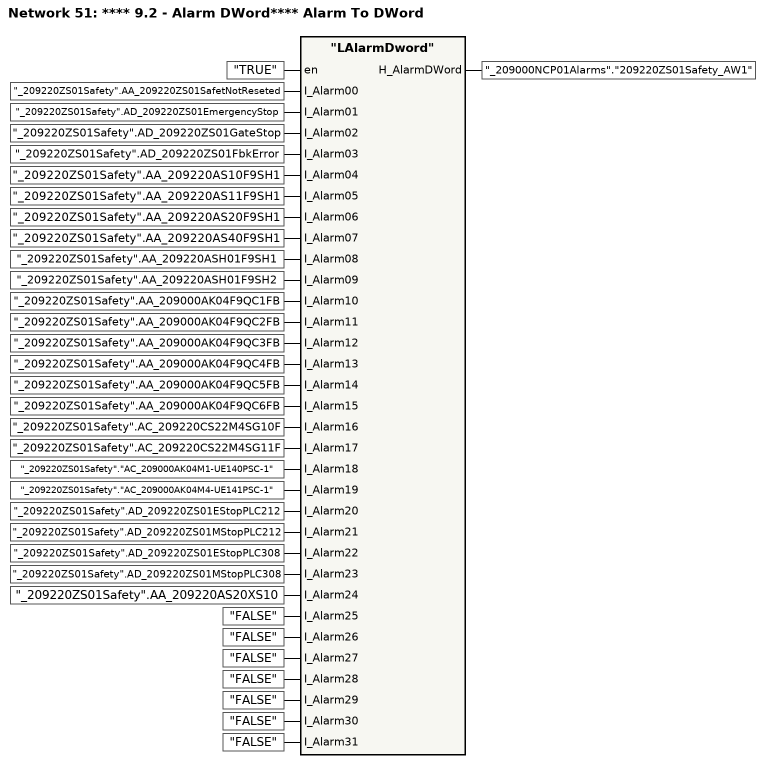
   IF "TRUE" THEN
       "LAlarmDword"(I_Alarm00 := "_209220ZS01Safety".AA_209220ZS01SafetNotReseted,
                     I_Alarm01 := "_209220ZS01Safety".AD_209220ZS01EmergencyStop,
                     I_Alarm02 := "_209220ZS01Safety".AD_209220ZS01GateStop,
                     I_Alarm03 := "_209220ZS01Safety".AD_209220ZS01FbkError,
                     I_Alarm04 := "_209220ZS01Safety".AA_209220AS10F9SH1,
                     I_Alarm05 := "_209220ZS01Safety".AA_209220AS11F9SH1,
                     I_Alarm06 := "_209220ZS01Safety".AA_209220AS20F9SH1,
                     I_Alarm07 := "_209220ZS01Safety".AA_209220AS40F9SH1,
                     I_Alarm08 := "_209220ZS01Safety".AA_209220ASH01F9SH1,
                     I_Alarm09 := "_209220ZS01Safety".AA_209220ASH01F9SH2,
                     I_Alarm10 := "_209220ZS01Safety".AA_209000AK04F9QC1FB,
                     I_Alarm11 := "_209220ZS01Safety".AA_209000AK04F9QC2FB,
                     I_Alarm12 := "_209220ZS01Safety".AA_209000AK04F9QC3FB,
                     I_Alarm13 := "_209220ZS01Safety".AA_209000AK04F9QC4FB,
                     I_Alarm14 := "_209220ZS01Safety".AA_209000AK04F9QC5FB,
                     I_Alarm15 := "_209220ZS01Safety".AA_209000AK04F9QC6FB,
                     I_Alarm16 := "_209220ZS01Safety".AC_209220CS22M4SG10F,
                     I_Alarm17 := "_209220ZS01Safety".AC_209220CS22M4SG11F,
                     I_Alarm18 := "_209220ZS01Safety"."AC_209000AK04M1-UE140PSC-1",
                     I_Alarm19 := "_209220ZS01Safety"."AC_209000AK04M4-UE141PSC-1",
                     I_Alarm20 := "_209220ZS01Safety".AD_209220ZS01EStopPLC212,
                     I_Alarm21 := "_209220ZS01Safety".AD_209220ZS01MStopPLC212,
                     I_Alarm22 := "_209220ZS01Safety".AD_209220ZS01EStopPLC308,
                     I_Alarm23 := "_209220ZS01Safety".AD_209220ZS01MStopPLC308,
                     I_Alarm24 := "_209220ZS01Safety".AA_209220AS20XS10,
                     I_Alarm25 := "FALSE",
                     I_Alarm26 := "FALSE",
                     I_Alarm27 := "FALSE",
                     I_Alarm28 := "FALSE",
                     I_Alarm29 := "FALSE",
                     I_Alarm30 := "FALSE",
                     I_Alarm31 := "FALSE",
                     H_AlarmDWord => "_209000NCP01Alarms"."209220ZS01Safety_AW1");
   END_IF;
END_REGION
END_FUNCTION
